FUNCTION_BLOCK FixedSchedule_FillerRoom
VAR_INPUT
	FillerRoom: STRING;
END_VAR

VAR_OUTPUT
	Scheduled_FixedHours: BOOL;
END_VAR
	
VAR
	total_minutes: INT;
	fbTime : FB_LocalSystemTime;
    stTime : TIMESTRUCT;
	Current_Hours: WORD; 
	Current_Minutes: WORD;
	
END_VAR

//Current time
fbTime(
    sNetID := '',
    bEnable := TRUE,
    dwCycle := 1000
);

stTime := fbTime.systemTime;
Current_Hours :=  stTime.wHour;
Current_Minutes := stTime.wMinute;


total_minutes := (WORD_TO_INT(Current_Hours) * 60) +
                  WORD_TO_INT(Current_Minutes);

// Shift per Filler Room
IF FillerRoom = 'FRA' OR FillerRoom = 'FRD'THEN
	Scheduled_FixedHours:= NOT((total_minutes>=120)AND(total_minutes<360)); //02:00am to 05:59 //(add 20 min after 2:00am just in case)
ELSIF  FillerRoom = 'FRC' THEN
	Scheduled_FixedHours:= NOT((total_minutes>=150)AND(total_minutes<390)); //02:30am to 06:29 //(add 20 min after 2:30am just in case)
ELSE
	Scheduled_FixedHours:= FALSE;
END_IF;

END_FUNCTION_BLOCK

(* stored: Version 1.1.0.1, ProductVersion 3.1.4024.15
   POU FixedSchedule_FillerRoom: Id {ae2c60b3-652d-4349-a466-bb31f628698b}, SpecialFunc None *)
